// SIMATIC S7-200 project (STEP 7-Micro/WIN), CPU 221 REL 01.10

ORGANIZATION_BLOCK 主程序:OB1
TITLE=程序注释
BEGIN
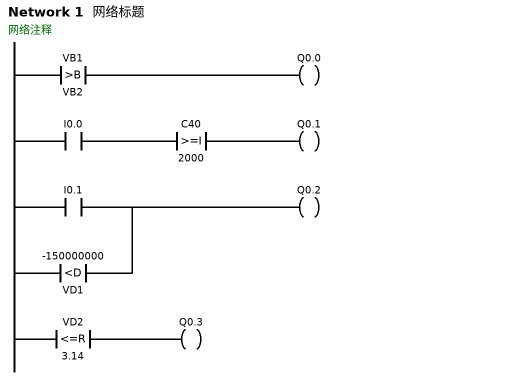
Network 1 // 网络标题
// 网络注释
// (network saved uncompiled; LAD cells follow)
// row 0: c0 -|>B|- VB1, VB2  c1 --  c2 -( ) Q0.0
// row 1: c0 -| |- I0.0  c1 -|>=I|- C40, 2000  c2 -( ) Q0.1
// row 2: c0 -| |- I0.1 v  c1 --  c2 -( ) Q0.2
// row 3: c0 -|<D|- -150000000, VD1 ^
// row 4: c0 -|<=R|- VD2, 3.14  c1 -( ) Q0.3
END_ORGANIZATION_BLOCK
